{attribute 'GeneratedUsingTerminal: EL6930-0000-0016'}
{attribute addProperty BoxType "EL6930-0000-0016"}
{attribute addProperty Description "EL6930, TwinSAFE PLC "}
{attribute addProperty Physics "KK"}
{attribute addProperty Id "DEVICE_InputsAT %I*DEVICE_Inputs_745C19EA6DEVICE_OutputsAT %Q*DEVICE_Outputs_DAFD38E02WcStateAT %I*WcState_9091E0EB2InfoDataAT %I*InfoData_32EB74EA10"}
{attribute addProperty CRC "191709189"}
{attribute addProperty Size "20"}
TYPE EL6930_0B6D4005 EXTENDS EtcSlaveTerminalBase_947E5A46 :
STRUCT
	{attribute addProperty Name "DEVICE_Inputs"}
	DEVICE_Inputs : DEVICE_Inputs_745C19EA;
	{attribute addProperty Name "DEVICE_Outputs"}
	DEVICE_Outputs : DEVICE_Outputs_DAFD38E0;
	{attribute addProperty Name "WcState"}
	WcState : WcState_9091E0EB;
	{attribute addProperty Name "InfoData"}
	InfoData : InfoData_32EB74EA;
END_STRUCT
END_TYPE

(* stored: Version 1.2.0.0, ProductVersion 3.1.4024.9
   DUT EL6930_0B6D4005: Id {bbff86a2-c6b5-4623-a61b-b0cc5a432b5a} *)
